PROGRAM prgUV
VAR
	fbUV1_1					: FB_EM_Electric_3P_Ext_Input;
	fbUV1_2					: FB_EM_Electric_3P_Ext_Input;
	fbUV2_1					: FB_EM_Electric_3P_Ext_Input;
	fbUV2_2					: FB_EM_Electric_3P_Ext_Input;
	fbUV2_3					: FB_EM_Electric_3P_Ext_Input;
	fbUV2_4					: FB_EM_Electric_3P_Ext_Input;
	fbUV3_1					: FB_EM_Electric_3P_Ext_Input;
	fbUV3_2					: FB_EM_Electric_3P_Ext_Input;
	fbUV3_3					: FB_EM_Electric_3P_Ext_Input;
	fbUV3_4					: FB_EM_Electric_3P_Ext_Input;
	timError_UV1_1			: TON;
	timError_UV1_2			: TON;
	timError_UV2_1			: TON;
	timError_UV2_2			: TON;
	timError_UV2_3			: TON;
	timError_UV2_4			: TON;
	timError_UV3_1			: TON;
	timError_UV3_2			: TON;
	timError_UV3_3			: TON;
	timError_UV3_4			: TON;
END_VAR

//UV1.1 for Limit Fuse Line (110kW)
//Error
IF prgCS11.byErrorWarningUV1_7 = 2 AND prgCS11.byErrorWarningUV1_8 = 2 THEN
	timError_UV1_1.IN := TRUE;
ELSE
	timError_UV1_1.IN := FALSE;
END_IF
	timError_UV1_1(IN:= , PT:= T#10S, Q=> , ET=> );

//Power from CS
fbUV1_1.lrPowerTotal := prgCS11.lrPowerUV1_7 + prgCS11.lrPowerUV1_8;
	fbUV1_1.lrPowerTotal := fbUV1_1.lrPowerTotal * 1000;

fbUV1_1(
	bEnable:= TRUE, 
	bPowerDataInvers:= , 
	bErrorExt:= timError_UV1_1.Q, 
	bWarningExt:= FALSE, 
	lrTotalCounterEnergy_Consumption:= 0, 
	lrTotalCounterEnergy_Production:= 0, 
	lrCounterEnergyT1_Consumption:= 0, 
	lrCounterEnergyT2_Consumption:= 0, 
	lrCounterEnergyT1_Production:= 0, 
	lrCounterEnergyT2_Production:= 0, 
	lrCurrentL1:= 0, 
	lrVoltageL1N:= 0, 
	lrVoltageL1L2:= 0, 
	lrPowerL1:= 0, 
	lrCurrentL2:= 0, 
	lrVoltageL2N:= 0, 
	lrVoltageL2L3:= 0, 
	lrPowerL2:= 0, 
	lrCurrentL3:= 0, 
	lrVoltageL3N:= 0, 
	lrVoltageL3L1:= 0, 
	lrPowerL3:= 0, 
	lrPowerTotal:= , 
	lrFrequency:= 0, 
	lrReactivePowerTotal:= 0, 
	lrApparentPowerTotal:= 0, 
	stDataEMPower=> , 
	stDataEMCounter=> , 
	diNrOfEM_OUT=> );
	
//UV1.2 for Limit Fuse Line (80kW)
//Error
IF prgCS11.byErrorWarningUV1_9 = 2 AND prgCS11.byErrorWarningUV1_10 = 2 AND prgCS12.byErrorWarningUV1_1 = 2 AND prgCS12.byErrorWarningUV1_2 = 2 AND prgCS12.byErrorWarningUV1_3 = 2 AND prgCS12.byErrorWarningUV1_4 = 2 AND prgCS12.byErrorWarningUV1_5 = 2 AND
	prgCS12.byErrorWarningUV1_6 = 2 THEN
		timError_UV1_2.IN := TRUE;
ELSE
		timError_UV1_2.IN := FALSE;
END_IF
	timError_UV1_2(IN:= , PT:= T#10S, Q=> , ET=> );

//Power from CS
fbUV1_2.lrPowerTotal := prgCS11.lrPowerUV1_9 + prgCS11.lrPowerUV1_10 + prgCS12.lrPowerUV1_1 + prgCS12.lrPowerUV1_2 + prgCS12.lrPowerUV1_3 + prgCS12.lrPowerUV1_4 + prgCS12.lrPowerUV1_5 + prgCS12.lrPowerUV1_6;
	fbUV1_2.lrPowerTotal := fbUV1_2.lrPowerTotal * 1000;

fbUV1_2(
	bEnable:= TRUE, 
	bPowerDataInvers:= , 
	bErrorExt:= timError_UV1_2.Q, 
	bWarningExt:= FALSE, 
	lrTotalCounterEnergy_Consumption:= 0, 
	lrTotalCounterEnergy_Production:= 0, 
	lrCounterEnergyT1_Consumption:= 0, 
	lrCounterEnergyT2_Consumption:= 0, 
	lrCounterEnergyT1_Production:= 0, 
	lrCounterEnergyT2_Production:= 0, 
	lrCurrentL1:= 0, 
	lrVoltageL1N:= 0, 
	lrVoltageL1L2:= 0, 
	lrPowerL1:= 0, 
	lrCurrentL2:= 0, 
	lrVoltageL2N:= 0, 
	lrVoltageL2L3:= 0, 
	lrPowerL2:= 0, 
	lrCurrentL3:= 0, 
	lrVoltageL3N:= 0, 
	lrVoltageL3L1:= 0, 
	lrPowerL3:= 0, 
	lrPowerTotal:= , 
	lrFrequency:= 0, 
	lrReactivePowerTotal:= 0, 
	lrApparentPowerTotal:= 0, 
	stDataEMPower=> , 
	stDataEMCounter=> , 
	diNrOfEM_OUT=> );
	
//UV2.1 for Limit Fuse Line (110kW)
//Error
IF prgCS6.byErrorWarningUV1_2 = 2 AND prgCS6.byErrorWarningUV1_3 = 2 AND prgCS6.byErrorWarningUV1_4 = 2 AND prgCS6.byErrorWarningUV1_5 = 2 AND prgCS6.byErrorWarningUV1_6 = 2 AND prgCS6.byErrorWarningUV1_7 = 2 AND prgCS6.byErrorWarningUV1_8 = 2 AND
	prgCS6.byErrorWarningUV1_9 = 2 AND prgCS6.byErrorWarningUV1_10 = 2 AND
		prgCS7.byErrorWarningUV1_1 = 2 AND prgCS7.byErrorWarningUV1_2 = 2 AND prgCS7.byErrorWarningUV1_3 = 2 AND prgCS7.byErrorWarningUV1_4 = 2 AND prgCS7.byErrorWarningUV1_5 = 2 THEN
			timError_UV2_1.IN := TRUE;
ELSE
			timError_UV2_1.IN := FALSE;
END_IF
	timError_UV2_1(IN:= , PT:= T#10S, Q=> , ET=> );

//Power from CS
fbUV2_1.lrPowerTotal := prgCS6.lrPowerUV1_2 + prgCS6.lrPowerUV1_3 + prgCS6.lrPowerUV1_4 + prgCS6.lrPowerUV1_5 + prgCS6.lrPowerUV1_6 + prgCS6.lrPowerUV1_7 + prgCS6.lrPowerUV1_8 + prgCS6.lrPowerUV1_9 + prgCS6.lrPowerUV1_10 +
							prgCS7.lrPowerUV1_1 + prgCS7.lrPowerUV1_2 + prgCS7.lrPowerUV1_3 + prgCS7.lrPowerUV1_4 + prgCS7.lrPowerUV1_5;
	fbUV2_1.lrPowerTotal := fbUV2_1.lrPowerTotal * 1000;	
							
fbUV2_1(
	bEnable:= TRUE, 
	bPowerDataInvers:= , 
	bErrorExt:= timError_UV2_1.Q, 
	bWarningExt:= FALSE, 
	lrTotalCounterEnergy_Consumption:= 0, 
	lrTotalCounterEnergy_Production:= 0, 
	lrCounterEnergyT1_Consumption:= 0, 
	lrCounterEnergyT2_Consumption:= 0, 
	lrCounterEnergyT1_Production:= 0, 
	lrCounterEnergyT2_Production:= 0, 
	lrCurrentL1:= 0, 
	lrVoltageL1N:= 0, 
	lrVoltageL1L2:= 0, 
	lrPowerL1:= 0, 
	lrCurrentL2:= 0, 
	lrVoltageL2N:= 0, 
	lrVoltageL2L3:= 0, 
	lrPowerL2:= 0, 
	lrCurrentL3:= 0, 
	lrVoltageL3N:= 0, 
	lrVoltageL3L1:= 0, 
	lrPowerL3:= 0, 
	lrPowerTotal:= , 
	lrFrequency:= 0, 
	lrReactivePowerTotal:= 0, 
	lrApparentPowerTotal:= 0, 
	stDataEMPower=> , 
	stDataEMCounter=> , 
	diNrOfEM_OUT=> );
	
//UV2.2 for Limit Fuse Line (110kW)
//Error
IF prgCS7.byErrorWarningUV1_6 = 2 AND prgCS7.byErrorWarningUV1_7 = 2 AND prgCS7.byErrorWarningUV1_8 = 2 AND prgCS7.byErrorWarningUV1_9 = 2 AND prgCS7.byErrorWarningUV1_10 = 2 AND
	prgCS8.byErrorWarningUV1_1 = 2 AND prgCS8.byErrorWarningUV1_2 = 2 AND prgCS8.byErrorWarningUV1_3 = 2 AND prgCS8.byErrorWarningUV1_4 = 2 AND prgCS8.byErrorWarningUV1_5 = 2 AND prgCS8.byErrorWarningUV1_6 = 2 THEN
		timError_UV2_2.IN := TRUE;
ELSE
		timError_UV2_2.IN := FALSE;
END_IF
	timError_UV2_2(IN:= , PT:= T#10S, Q=> , ET=> );

//Power from CS
fbUV2_2.lrPowerTotal := prgCS7.lrPowerUV1_6 + prgCS7.lrPowerUV1_7 + prgCS7.lrPowerUV1_8 + prgCS7.lrPowerUV1_9 + prgCS7.lrPowerUV1_10 +
							prgCS8.lrPowerUV1_1 + prgCS8.lrPowerUV1_2 + prgCS8.lrPowerUV1_3 + prgCS8.lrPowerUV1_4 + prgCS8.lrPowerUV1_5 + prgCS8.lrPowerUV1_6;
	fbUV2_2.lrPowerTotal := fbUV2_2.lrPowerTotal * 1000;
							
fbUV2_2(
	bEnable:= TRUE, 
	bPowerDataInvers:= , 
	bErrorExt:= timError_UV2_2.Q, 
	bWarningExt:= FALSE, 
	lrTotalCounterEnergy_Consumption:= 0, 
	lrTotalCounterEnergy_Production:= 0, 
	lrCounterEnergyT1_Consumption:= 0, 
	lrCounterEnergyT2_Consumption:= 0, 
	lrCounterEnergyT1_Production:= 0, 
	lrCounterEnergyT2_Production:= 0, 
	lrCurrentL1:= 0, 
	lrVoltageL1N:= 0, 
	lrVoltageL1L2:= 0, 
	lrPowerL1:= 0, 
	lrCurrentL2:= 0, 
	lrVoltageL2N:= 0, 
	lrVoltageL2L3:= 0, 
	lrPowerL2:= 0, 
	lrCurrentL3:= 0, 
	lrVoltageL3N:= 0, 
	lrVoltageL3L1:= 0, 
	lrPowerL3:= 0, 
	lrPowerTotal:= , 
	lrFrequency:= 0, 
	lrReactivePowerTotal:= 0, 
	lrApparentPowerTotal:= 0, 
	stDataEMPower=> , 
	stDataEMCounter=> , 
	diNrOfEM_OUT=> );
	
//UV2.3 for Limit Fuse Line (110kW)
//Error
IF prgCS8.byErrorWarningUV1_8 = 2 AND prgCS9.byErrorWarningUV1_2 = 2 AND prgCS9.byErrorWarningUV1_3 = 2 AND prgCS9.byErrorWarningUV1_6 = 2 AND prgCS9.byErrorWarningUV1_7 = 2 THEN
	timError_UV2_3.IN := TRUE;
ELSE
	timError_UV2_3.IN := FALSE;
END_IF
	timError_UV2_3(IN:= , PT:= T#10S, Q=> , ET=> );

//Power from CS
fbUV2_3.lrPowerTotal := prgCS8.lrPowerUV1_8 + prgCS9.lrPowerUV1_2 + prgCS9.lrPowerUV1_3 + prgCS9.lrPowerUV1_6 + prgCS9.lrPowerUV1_7;
	fbUV2_3.lrPowerTotal := fbUV2_3.lrPowerTotal * 1000;

fbUV2_3(
	bEnable:= TRUE, 
	bPowerDataInvers:= , 
	bErrorExt:= timError_UV2_3.Q, 
	bWarningExt:= FALSE, 
	lrTotalCounterEnergy_Consumption:= 0, 
	lrTotalCounterEnergy_Production:= 0, 
	lrCounterEnergyT1_Consumption:= 0, 
	lrCounterEnergyT2_Consumption:= 0, 
	lrCounterEnergyT1_Production:= 0, 
	lrCounterEnergyT2_Production:= 0, 
	lrCurrentL1:= 0, 
	lrVoltageL1N:= 0, 
	lrVoltageL1L2:= 0, 
	lrPowerL1:= 0, 
	lrCurrentL2:= 0, 
	lrVoltageL2N:= 0, 
	lrVoltageL2L3:= 0, 
	lrPowerL2:= 0, 
	lrCurrentL3:= 0, 
	lrVoltageL3N:= 0, 
	lrVoltageL3L1:= 0, 
	lrPowerL3:= 0, 
	lrPowerTotal:= , 
	lrFrequency:= 0, 
	lrReactivePowerTotal:= 0, 
	lrApparentPowerTotal:= 0, 
	stDataEMPower=> , 
	stDataEMCounter=> , 
	diNrOfEM_OUT=> );
	
//UV2.4 for Limit Fuse Line (110kW)
//Error
IF prgCS9.byErrorWarningUV1_10 = 2 AND prgCS10.byErrorWarningUV1_1 = 2 AND prgCS10.byErrorWarningUV1_2 = 2 AND prgCS10.byErrorWarningUV1_3 = 2 AND prgCS10.byErrorWarningUV1_4 = 2 AND prgCS10.byErrorWarningUV1_5 = 2 AND prgCS10.byErrorWarningUV1_6 = 2 AND
	prgCS10.byErrorWarningUV1_7 = 2 THEN
		timError_UV2_4.IN := TRUE;
ELSE
		timError_UV2_4.IN := FALSE;
END_IF
	timError_UV2_4(IN:= , PT:= T#10S, Q=> , ET=> );

//Power from CS
fbUV2_4.lrPowerTotal := prgCS9.lrPowerUV1_10 + prgCS10.lrPowerUV1_1 + prgCS10.lrPowerUV1_2 + prgCS10.lrPowerUV1_3 + prgCS10.lrPowerUV1_4 + prgCS10.lrPowerUV1_5 + prgCS10.lrPowerUV1_6 + prgCS10.lrPowerUV1_7;
	fbUV2_4.lrPowerTotal := fbUV2_4.lrPowerTotal * 1000;

fbUV2_4(
	bEnable:= TRUE, 
	bPowerDataInvers:= , 
	bErrorExt:= timError_UV2_4.Q, 
	bWarningExt:= FALSE, 
	lrTotalCounterEnergy_Consumption:= 0, 
	lrTotalCounterEnergy_Production:= 0, 
	lrCounterEnergyT1_Consumption:= 0, 
	lrCounterEnergyT2_Consumption:= 0, 
	lrCounterEnergyT1_Production:= 0, 
	lrCounterEnergyT2_Production:= 0, 
	lrCurrentL1:= 0, 
	lrVoltageL1N:= 0, 
	lrVoltageL1L2:= 0, 
	lrPowerL1:= 0, 
	lrCurrentL2:= 0, 
	lrVoltageL2N:= 0, 
	lrVoltageL2L3:= 0, 
	lrPowerL2:= 0, 
	lrCurrentL3:= 0, 
	lrVoltageL3N:= 0, 
	lrVoltageL3L1:= 0, 
	lrPowerL3:= 0, 
	lrPowerTotal:= , 
	lrFrequency:= 0, 
	lrReactivePowerTotal:= 0, 
	lrApparentPowerTotal:= 0, 
	stDataEMPower=> , 
	stDataEMCounter=> , 
	diNrOfEM_OUT=> );
	
//UV3.1 for Limit Fuse Line (110kW)
//Error
IF prgCS1.byErrorWarningUV1_1 = 2 AND prgCS1.byErrorWarningUV1_2 = 2 AND prgCS1.byErrorWarningUV1_3 = 2 AND prgCS1.byErrorWarningUV1_4 = 2 AND prgCS1.byErrorWarningUV1_5 = 2 AND prgCS1.byErrorWarningUV1_6 = 2 AND prgCS1.byErrorWarningUV1_7 = 2 AND
	prgCS1.byErrorWarningUV1_8 = 2 AND prgCS1.byErrorWarningUV1_9 = 2 AND prgCS1.byErrorWarningUV1_10 = 2 AND
		prgCS2.byErrorWarningUV1_1 = 2 AND prgCS2.byErrorWarningUV1_2 = 2 AND prgCS2.byErrorWarningUV1_3 = 2 AND prgCS2.byErrorWarningUV1_4 = 2 THEN
			timError_UV3_1.IN := TRUE;
ELSE
			timError_UV3_1.IN := FALSE;
END_IF
	timError_UV3_1(IN:= , PT:= T#10S, Q=> , ET=> );

//Power from CS
fbUV3_1.lrPowerTotal := prgCS1.lrPowerUV1_1 + prgCS1.lrPowerUV1_2 + prgCS1.lrPowerUV1_3 + prgCS1.lrPowerUV1_4 + prgCS1.lrPowerUV1_5 + prgCS1.lrPowerUV1_6 + prgCS1.lrPowerUV1_7 + prgCS1.lrPowerUV1_8 + prgCS1.lrPowerUV1_9 + prgCS1.lrPowerUV1_10 +
							prgCS2.lrPowerUV1_1 + prgCS2.lrPowerUV1_2 + prgCS2.lrPowerUV1_3 + prgCS2.lrPowerUV1_4;
	fbUV3_1.lrPowerTotal := fbUV3_1.lrPowerTotal * 1000;
							
fbUV3_1(
	bEnable:= TRUE, 
	bPowerDataInvers:= , 
	bErrorExt:= timError_UV3_1.Q, 
	bWarningExt:= FALSE, 
	lrTotalCounterEnergy_Consumption:= 0, 
	lrTotalCounterEnergy_Production:= 0, 
	lrCounterEnergyT1_Consumption:= 0, 
	lrCounterEnergyT2_Consumption:= 0, 
	lrCounterEnergyT1_Production:= 0, 
	lrCounterEnergyT2_Production:= 0, 
	lrCurrentL1:= 0, 
	lrVoltageL1N:= 0, 
	lrVoltageL1L2:= 0, 
	lrPowerL1:= 0, 
	lrCurrentL2:= 0, 
	lrVoltageL2N:= 0, 
	lrVoltageL2L3:= 0, 
	lrPowerL2:= 0, 
	lrCurrentL3:= 0, 
	lrVoltageL3N:= 0, 
	lrVoltageL3L1:= 0, 
	lrPowerL3:= 0, 
	lrPowerTotal:= , 
	lrFrequency:= 0, 
	lrReactivePowerTotal:= 0, 
	lrApparentPowerTotal:= 0, 
	stDataEMPower=> , 
	stDataEMCounter=> , 
	diNrOfEM_OUT=> );
	
//UV3.2 for Limit Fuse Line (80kW)
//Error
IF prgCS2.byErrorWarningUV1_5 = 2 AND prgCS2.byErrorWarningUV1_6 = 2 AND prgCS2.byErrorWarningUV1_7 = 2 AND prgCS2.byErrorWarningUV1_8 = 2 AND prgCS2.byErrorWarningUV1_9 = 2 AND prgCS2.byErrorWarningUV1_10 = 2 AND
	prgCS3.byErrorWarningUV1_1 = 2 AND prgCS3.byErrorWarningUV1_2 = 2 AND prgCS3.byErrorWarningUV1_3 = 2 AND prgCS3.byErrorWarningUV1_4 = 2 AND prgCS3.byErrorWarningUV1_5 = 2 AND prgCS3.byErrorWarningUV1_6 = 2 THEN
		timError_UV3_2.IN := TRUE;
ELSE
		timError_UV3_2.IN := FALSE;
END_IF
	timError_UV3_2(IN:= , PT:= T#10S, Q=> , ET=> );

//Power from CS
fbUV3_2.lrPowerTotal := prgCS2.lrPowerUV1_5 + prgCS2.lrPowerUV1_6 + prgCS2.lrPowerUV1_7 + prgCS2.lrPowerUV1_8 + prgCS2.lrPowerUV1_9 + prgCS2.lrPowerUV1_10 +
							prgCS3.lrPowerUV1_1 + prgCS3.lrPowerUV1_2 + prgCS3.lrPowerUV1_3 + prgCS3.lrPowerUV1_4 + prgCS3.lrPowerUV1_5 + prgCS3.lrPowerUV1_6;
	fbUV3_2.lrPowerTotal := fbUV3_2.lrPowerTotal * 1000;
							
fbUV3_2(
	bEnable:= TRUE, 
	bPowerDataInvers:= , 
	bErrorExt:= timError_UV3_2.Q, 
	bWarningExt:= FALSE, 
	lrTotalCounterEnergy_Consumption:= 0, 
	lrTotalCounterEnergy_Production:= 0, 
	lrCounterEnergyT1_Consumption:= 0, 
	lrCounterEnergyT2_Consumption:= 0, 
	lrCounterEnergyT1_Production:= 0, 
	lrCounterEnergyT2_Production:= 0, 
	lrCurrentL1:= 0, 
	lrVoltageL1N:= 0, 
	lrVoltageL1L2:= 0, 
	lrPowerL1:= 0, 
	lrCurrentL2:= 0, 
	lrVoltageL2N:= 0, 
	lrVoltageL2L3:= 0, 
	lrPowerL2:= 0, 
	lrCurrentL3:= 0, 
	lrVoltageL3N:= 0, 
	lrVoltageL3L1:= 0, 
	lrPowerL3:= 0, 
	lrPowerTotal:= , 
	lrFrequency:= 0, 
	lrReactivePowerTotal:= 0, 
	lrApparentPowerTotal:= 0, 
	stDataEMPower=> , 
	stDataEMCounter=> , 
	diNrOfEM_OUT=> );
	
//UV3.3 for Limit Fuse Line (110kW)
//Error
IF prgCS3.byErrorWarningUV1_7 = 2 AND prgCS3.byErrorWarningUV1_8 = 2 AND prgCS3.byErrorWarningUV1_9 = 2 AND prgCS3.byErrorWarningUV1_10 = 2 AND
	prgCS4.byErrorWarningUV1_1 = 2 AND prgCS4.byErrorWarningUV1_2 = 2 AND prgCS4.byErrorWarningUV1_3 = 2 AND prgCS4.byErrorWarningUV1_4 = 2 AND prgCS4.byErrorWarningUV1_5 = 2 AND prgCS4.byErrorWarningUV1_6 = 2 AND prgCS4.byErrorWarningUV1_7 = 2 AND
		prgCS4.byErrorWarningUV1_8 = 2 THEN
			timError_UV3_3.IN := TRUE;
ELSE
			timError_UV3_3.IN := FALSE;
END_IF
	timError_UV3_3(IN:= , PT:= T#10S, Q=> , ET=> );

//Power from CS
fbUV3_3.lrPowerTotal := prgCS3.lrPowerUV1_7 + prgCS3.lrPowerUV1_8 + prgCS3.lrPowerUV1_9 + prgCS3.lrPowerUV1_10 +
							prgCS4.lrPowerUV1_1 + prgCS4.lrPowerUV1_2 + prgCS4.lrPowerUV1_3 + prgCS4.lrPowerUV1_4 + prgCS4.lrPowerUV1_5 + prgCS4.lrPowerUV1_6 + prgCS4.lrPowerUV1_7 + prgCS4.lrPowerUV1_8;
	fbUV3_3.lrPowerTotal := fbUV3_3.lrPowerTotal * 1000;
							
fbUV3_3(
	bEnable:= TRUE, 
	bPowerDataInvers:= , 
	bErrorExt:= timError_UV3_3.Q, 
	bWarningExt:= FALSE, 
	lrTotalCounterEnergy_Consumption:= 0, 
	lrTotalCounterEnergy_Production:= 0, 
	lrCounterEnergyT1_Consumption:= 0, 
	lrCounterEnergyT2_Consumption:= 0, 
	lrCounterEnergyT1_Production:= 0, 
	lrCounterEnergyT2_Production:= 0, 
	lrCurrentL1:= 0, 
	lrVoltageL1N:= 0, 
	lrVoltageL1L2:= 0, 
	lrPowerL1:= 0, 
	lrCurrentL2:= 0, 
	lrVoltageL2N:= 0, 
	lrVoltageL2L3:= 0, 
	lrPowerL2:= 0, 
	lrCurrentL3:= 0, 
	lrVoltageL3N:= 0, 
	lrVoltageL3L1:= 0, 
	lrPowerL3:= 0, 
	lrPowerTotal:= , 
	lrFrequency:= 0, 
	lrReactivePowerTotal:= 0, 
	lrApparentPowerTotal:= 0, 
	stDataEMPower=> , 
	stDataEMCounter=> , 
	diNrOfEM_OUT=> );
	
//UV3.4 for Limit Fuse Line (110kW)
//Error
IF prgCS4.byErrorWarningUV1_9 = 2 AND prgCS4.byErrorWarningUV1_10 = 2 AND
	prgCS5.byErrorWarningUV1_1 = 2 AND prgCS5.byErrorWarningUV1_2 = 2 AND prgCS5.byErrorWarningUV1_3 = 2 AND prgCS5.byErrorWarningUV1_4 = 2 AND prgCS5.byErrorWarningUV1_5 = 2 AND prgCS5.byErrorWarningUV1_6 = 2 AND prgCS5.byErrorWarningUV1_7 = 2 AND
		prgCS5.byErrorWarningUV1_8 = 2 THEN
			timError_UV3_4.IN := TRUE;
ELSE
			timError_UV3_4.IN := FALSE;
END_IF
	timError_UV3_4(IN:= , PT:= T#10S, Q=> , ET=> );

//Power from CS
fbUV3_4.lrPowerTotal := prgCS4.lrPowerUV1_9 + prgCS4.lrPowerUV1_10 +
							prgCS5.lrPowerUV1_1 + prgCS5.lrPowerUV1_2 + prgCS5.lrPowerUV1_3 + prgCS5.lrPowerUV1_4 + prgCS5.lrPowerUV1_5 + prgCS5.lrPowerUV1_6 + prgCS5.lrPowerUV1_7 + prgCS5.lrPowerUV1_8;
	fbUV3_4.lrPowerTotal := fbUV3_4.lrPowerTotal * 1000;
							
fbUV3_4(
	bEnable:= TRUE, 
	bPowerDataInvers:= , 
	bErrorExt:= timError_UV3_4.Q, 
	bWarningExt:= FALSE, 
	lrTotalCounterEnergy_Consumption:= 0, 
	lrTotalCounterEnergy_Production:= 0, 
	lrCounterEnergyT1_Consumption:= 0, 
	lrCounterEnergyT2_Consumption:= 0, 
	lrCounterEnergyT1_Production:= 0, 
	lrCounterEnergyT2_Production:= 0, 
	lrCurrentL1:= 0, 
	lrVoltageL1N:= 0, 
	lrVoltageL1L2:= 0, 
	lrPowerL1:= 0, 
	lrCurrentL2:= 0, 
	lrVoltageL2N:= 0, 
	lrVoltageL2L3:= 0, 
	lrPowerL2:= 0, 
	lrCurrentL3:= 0, 
	lrVoltageL3N:= 0, 
	lrVoltageL3L1:= 0, 
	lrPowerL3:= 0, 
	lrPowerTotal:= , 
	lrFrequency:= 0, 
	lrReactivePowerTotal:= 0, 
	lrApparentPowerTotal:= 0, 
	stDataEMPower=> , 
	stDataEMCounter=> , 
	diNrOfEM_OUT=> );

END_PROGRAM

(* stored: Version 1.1.0.1, ProductVersion 3.1.4024.9
   POU prgUV: Id {54849f6e-b57c-46bf-9186-df090c664b9a}, SpecialFunc None *)
